TYPE SCRIPTNAME :
STRUCT
	payload		:T_MaxString;	
	start		:BOOL	:= FALSE;
	end			:BOOL	:= FALSE;		
END_STRUCT
END_TYPE

(* stored: Version 1.1.0.1, ProductVersion 3.1.4026.18
   DUT SCRIPTNAME: Id {349cd820-c227-46b8-b9df-7e626fc5d05c} *)
